Staubli VAL3: list.pgx

program list(string pTitle (dimensions=1), num pX (dimensions=1), num pY (dimensions=1), num pDx (dimensions=1), num pDy (dimensions=1), string& sName[] (dimensions=1))
  local num lDx
  local num lDy
  local num lI
  local num lJ
  local string lStr
  local string lStrLine
  local num lValue
  local num l_nsize
begin
  //-----------------------------------------------------------------------
  //Header begin
  //Description of program
  //  在列pX和行pY处创建宽pDx，高pDy的列表；列表名称pTitle；列表内容为sName
  //Input parameters
  //  string pTitle:列表名
  //  num pX: 列表左上角列位置
  //  num PY: 列表左上角行位置
  //  num pDx: 列表宽
  //  num pDy：列表高
  //  string sName:列表显示内容
  //Output paramaters
  //
  //Example
  //  call list("list1",10,0,20,20)
  //Creation : 2012-06-11 - PF.Zhong
  //Header end
  //-----------------------------------------------------------------------
  //
  lStrLine="─────────────────────────────────────────"
  lDx=pDx
  lDy=pDy
  l_nsize=size(sName)
  //Top
  lStr="┌"+mid(lStrLine,lDx,0)+"┐"
  gotoxy(pX,pY)
  put(lStr)
  lValue=pX+2
  //Title
  if pTitle!=""
    call leftPos("┤"+pTitle+"├",lDx,pTitle)
    gotoxy(pX+lDx-getDisplayLen(pTitle)+1,pY)
    put(pTitle)
  endIf
  //Containt
  for lJ=1 to lDy
    lValue=pY+lJ
    lStr="│"
    gotoxy(pX,lValue)
    put(lStr)
    if lJ<=l_nsize
      if sName[lJ-1]!=""
        put(sName[lJ-1])
      endIf
    endIf
    gotoxy(pX+lDx+1,lValue)
    put(lStr)
  endFor
  //Bottom
  lValue=pY+lJ
  lStr="└"+mid(lStrLine,lDx,0)+"┘"
  gotoxy(pX,lValue)
  put(lStr)
end
